Fanuc KAREL source: ka00090.KL

-- PROVISIONAL review KL for V770-1; original PC SHA256 0116c2af34009bb8bfded76657b9aa06081271eaa7a8a0d8a405c63fae52aaae
-- Incomplete behavior may be omitted. Consult companion uncertainty JSON. Do not deploy.
PROGRAM KA00090
%NOLOCKGROUP
-- UNRESOLVED_DECL SRC type=000199
-- UNRESOLVED_DECL DST type=000102
BEGIN
  -- UNRESOLVED_PC offsets 5-25; opcodes 49,7E,4A
  -- UNRESOLVED_PC offsets 30-34; opcodes 7F
END KA00090
